PROGRAM PRG_1_PlcTask
VAR
END_VAR

PRG_2_PMPS_POST();
PRG_MR1K3_SOMS();
PRG_MR2K3_SOMS();

END_PROGRAM

(* stored: Version 1.1.0.1, ProductVersion 3.1.4024.12
   POU PRG_1_PlcTask: Id {d2db6153-7cba-41a1-b567-1fc62a8f9d77}, SpecialFunc None *)
